// TIA Portal project "Modbus_ESP32_1212SIPLUS" (V19)

(* hardware
DEVICE "S7-1200 station_1"  S7-1200 Station
   slot 0: "Rack_0"  S7-1200 Rack  Rack  V1.0
   slot 1: "PLC_2"  CPU 1212C DC/DC/DC  6ES7 212-1AE31-0XB0  V3.0
*)

// ===== PLC "PLC_2"  CPU 1212C DC/DC/DC =====

DATA_BLOCK "Data"   // DB2
{ S7_Optimized_Access := 'FALSE' }
VERSION : 0.1
   VAR
      holdReg : Array[0..9] of Int;
   END_VAR
BEGIN
END_DATA_BLOCK

DATA_BLOCK "Main_iDB"   // DB1050
{ S7_Optimized_Access := 'TRUE' }
VERSION : 0.1
// stored: InstanceOfName FB_Main
"FB_Main"
BEGIN
END_DATA_BLOCK

FUNCTION_BLOCK "FB_Main"   // FB1000, FBD
{ S7_Optimized_Access := 'TRUE' }
VERSION : 0.1
   VAR
      MB_SERVER : MB_SERVER;
   END_VAR
BEGIN

REGION Network 1
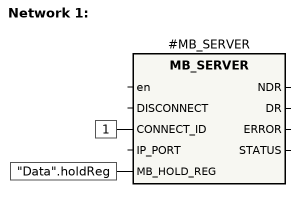
   #MB_SERVER(CONNECT_ID := 1, MB_HOLD_REG := "Data".holdReg);   // MB_SERVER
END_REGION
END_FUNCTION_BLOCK

ORGANIZATION_BLOCK "Main"   // OB1, LAD, ProgramCycle
TITLE = "Main Program Sweep (Cycle)"
{ S7_Optimized_Access := 'TRUE' }
VERSION : 0.1
BEGIN

REGION Network 1
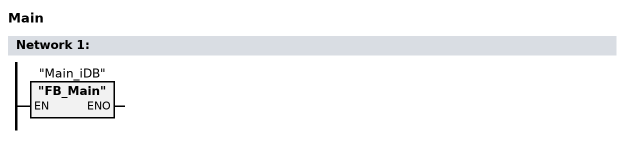
   RUNG wire#powerrail
      "Main_iDB"()
   END_RUNG
   // the same network as SCL:
   "Main_iDB"();   // "FB_Main"
END_REGION
END_ORGANIZATION_BLOCK